// TIA Portal V18 export
DATA_BLOCK "WebDB"   // DB5
{ S7_Optimized_Access := 'FALSE' }
VERSION : 0.1
// stored: AutoNumber true, DBAccessibleFromOPCUA true, IsOnlyStoredInLoadMemory false, IsWriteProtectedInAS false
   VAR
      Enabled_Devices : Bool;   // Diagnostic value, necessary in step 3 (Check if system is ready); TRUE if OK;
      Ready_Devices : Bool;   // Diagnostic value, necessary in step 3 (Check if system is ready); TRUE if OK;
      Warning_Devices : Bool;   // Diagnostic value, necessary in step 3 (Check if system is ready); TRUE if OK;
      Fault_Devices : Bool;   // Diagnostic value, necessary in step 3 (Check if system is ready); TRUE if OK;
      diagMode { ExternalAccessible := 'False'; ExternalVisible := 'False'; ExternalWritable := 'False'} : UInt := 1;   // Diagnostic mode : 0
      myLADDR { ExternalAccessible := 'False'; ExternalVisible := 'False'; ExternalWritable := 'False'} : HW_ANY := 52;   // ID of CPUExecutUnit : 52 PLC ID: 64
      returnValue : Int;   // No error: 0
      CountDiagDetails : UInt;   // Should always be 0
      PLCDiag { S7_SetPoint := 'True'} : DIS;   // Read value of diagnostic
      Start_Machine : Bool;   // Button - Start Machine
      Stop_Machine : Bool;   // Button - Stop Machine
      Reset_error { ExternalAccessible := 'False'; ExternalVisible := 'False'; ExternalWritable := 'False'} : Bool;   // Button - Reset error after emergancy stop and other situation
      Stop_All_Axis : Bool;
      XInput : Struct
         EnableDrive : Bool;
         Stop : Bool;
         Halt : Bool;
         Brake : Bool;
         ResetFault : Bool;
         HMIAccessLocked : Bool;
         OPM : Int;   // Operating Mode ???
         StartTask : Bool;
         StartHoming : Bool;
         JogPos : Bool;
         JogNeg : Bool;
         TeachActValue : Bool;
         ClearRemPos : Bool;
         Relative : Bool;
         DeactivateStrokeLimit : Bool;
         ExecuteFunction : Bool;
         RecordNo : Int;
         SetFunctionNumber : Int;
         SetFunctionGroup : Int;
         SetValueVelocity : DInt := 20;
         SetValuePosition : DInt;
         SetValueForceRamp : DInt;
         SetValueForce : DInt;
         SetValueRotRamp : DInt;
         SetValueRotSpeed : DInt;
      END_STRUCT;
      XOutput : Struct
         DriveEnabled : Bool;
         Ready : Bool;
         Warning : Bool;
         Fault : Bool;
         SupplyVoltPresent : Bool;
         ControlFCT_HMI : Bool;
         StateOPM : Int;
         HaltNotActive : Bool;
         AckStart : Bool;
         MC : Bool;
         AckTeach : Bool;
         DriveMoving : Bool;
         DragError : Bool;
         StandStillControl : Bool;
         HomingValid : Bool;
         ActualRecordNo : Int;
         RC1 : Bool;
         RCC : Bool;
         VelocityLimitReached : Bool;
         StrokeLimitReached : Bool;
         FunctionIsActive : Bool;
         ActualFunctionNumber : Int;
         ActualFunctionGroup : Int;
         ActualPosition : DInt;
         ActualVelocity : DInt;
         ActualForce : DInt;
         ActualRotRamp : DInt;
         ActualRotSpeed : DInt;
      END_STRUCT;
      XAddOn1 : Struct
         XTargetRange : DInt := 1000;
         XTargetReached : Bool;
         XOverrange : Bool;
         Error_message_X : DInt;   // Number of error in DINT. Check error in CMMP documentation
         Restart_CMMO_X : Bool;   // Restart CMMP X controller
      END_STRUCT;
      YInput : Struct
         EnableDrive : Bool;
         Stop : Bool;
         Halt : Bool;
         Brake : Bool;
         ResetFault : Bool;
         HMIAccessLocked : Bool;
         OPM : Int;   // Operating Mode ???
         StartTask : Bool;
         StartHoming : Bool;
         JogPos : Bool;
         JogNeg : Bool;
         TeachActValue : Bool;
         ClearRemPos : Bool;
         Relative : Bool;
         DeactivateStrokeLimit : Bool;
         ExecuteFunction : Bool;
         RecordNo : Int;
         SetFunctionNumber : Int;
         SetFunctionGroup : Int;
         SetValueVelocity : DInt := 20;
         SetValuePosition : DInt;
         SetValueForceRamp : DInt;
         SetValueForce : DInt;
         SetValueRotRamp : DInt;
         SetValueRotSpeed : DInt;
      END_STRUCT;
      YOutput : Struct
         DriveEnabled : Bool;
         Ready : Bool;
         Warning : Bool;
         Fault : Bool;
         SupplyVoltPresent : Bool;
         ControlFCT_HMI : Bool;
         StateOPM : Int;
         HaltNotActive : Bool;
         AckStart : Bool;
         MC : Bool;
         AckTeach : Bool;
         DriveMoving : Bool;
         DragError : Bool;
         StandStillControl : Bool;
         HomingValid : Bool;
         ActualRecordNo : Int;
         RC1 : Bool;
         RCC : Bool;
         VelocityLimitReached : Bool;
         StrokeLimitReached : Bool;
         FunctionIsActive : Bool;
         ActualFunctionNumber : Int;
         ActualFunctionGroup : Int;
         ActualPosition : DInt;
         ActualVelocity : DInt;
         ActualForce : DInt;
         ActualRotRamp : DInt;
         ActualRotSpeed : DInt;
      END_STRUCT;
      YAddOn1 : Struct
         YTargetRange : DInt := 1000;
         YTargetReached : Bool;
         YOverrange : Bool;
         Error_message_Y : DInt;   // Number of error in DINT. Check error in CMMP documentation
         Restart_CMMO_Y : Bool;   // Restart CMMP Y controller
      END_STRUCT;
      Z1Input : Struct
         EnableDrive : Bool;
         Stop : Bool;
         Halt : Bool;
         Brake : Bool;
         ResetFault : Bool;
         HMIAccessLocked : Bool;
         OPM : Int;   // Operating Mode ???
         StartTask : Bool;
         StartHoming : Bool;
         JogPos : Bool;
         JogNeg : Bool;
         TeachActValue : Bool;
         ClearRemPos : Bool;
         Relative : Bool;
         DeactivateStrokeLimit : Bool;
         ExecuteFunction : Bool;
         RecordNo : Int;
         SetFunctionNumber : Int;
         SetFunctionGroup : Int;
         SetValueVelocity : DInt := 20;
         SetValuePosition : DInt;
         SetValueForceRamp : DInt;
         SetValueForce : DInt;
         SetValueRotRamp : DInt;
         SetValueRotSpeed : DInt;
      END_STRUCT;
      Z1Output : Struct
         DriveEnabled : Bool;
         Ready : Bool;
         Warning : Bool;
         Fault : Bool;
         SupplyVoltPresent : Bool;
         ControlFCT_HMI : Bool;
         StateOPM : Int;
         HaltNotActive : Bool;
         AckStart : Bool;
         MC : Bool;
         AckTeach : Bool;
         DriveMoving : Bool;
         DragError : Bool;
         StandStillControl : Bool;
         HomingValid : Bool;
         ActualRecordNo : Int;
         RC1 : Bool;
         RCC : Bool;
         VelocityLimitReached : Bool;
         StrokeLimitReached : Bool;
         FunctionIsActive : Bool;
         ActualFunctionNumber : Int;
         ActualFunctionGroup : Int;
         ActualPosition : DInt;
         ActualVelocity : DInt;
         ActualForce : DInt;
         ActualRotRamp : DInt;
         ActualRotSpeed : DInt;
      END_STRUCT;
      Z1AddOn1 : Struct
         Z1TargetRange : DInt := 1000;
         Z1TargetReached : Bool;
         Z1Overrange : Bool;
         Error_message_Z1 : DInt;   // Number of error in DINT. Check error in CMMO documentation
         Restart_CMMO_Z1 : Bool;   // Restart CMMO Z1 controller
      END_STRUCT;
      Z2Input : Struct
         EnableDrive : Bool;
         Stop : Bool;
         Halt : Bool;
         Brake : Bool;
         ResetFault : Bool;
         HMIAccessLocked : Bool;
         OPM : Int;   // Operating Mode ???
         StartTask : Bool;
         StartHoming : Bool;
         JogPos : Bool;
         JogNeg : Bool;
         TeachActValue : Bool;
         ClearRemPos : Bool;
         Relative : Bool;
         DeactivateStrokeLimit : Bool;
         ExecuteFunction : Bool;
         RecordNo : Int;
         SetFunctionNumber : Int;
         SetFunctionGroup : Int;
         SetValueVelocity : DInt := 20;
         SetValuePosition : DInt;
         SetValueForceRamp : DInt;
         SetValueForce : DInt;
         SetValueRotRamp : DInt;
         SetValueRotSpeed : DInt;
      END_STRUCT;
      Z2Output : Struct
         DriveEnabled : Bool;
         Ready : Bool;
         Warning : Bool;
         Fault : Bool;
         SupplyVoltPresent : Bool;
         ControlFCT_HMI : Bool;
         StateOPM : Int;
         HaltNotActive : Bool;
         AckStart : Bool;
         MC : Bool;
         AckTeach : Bool;
         DriveMoving : Bool;
         DragError : Bool;
         StandStillControl : Bool;
         HomingValid : Bool;
         ActualRecordNo : Int;
         RC1 : Bool;
         RCC : Bool;
         VelocityLimitReached : Bool;
         StrokeLimitReached : Bool;
         FunctionIsActive : Bool;
         ActualFunctionNumber : Int;
         ActualFunctionGroup : Int;
         ActualPosition : DInt;
         ActualVelocity : DInt;
         ActualForce : DInt;
         ActualRotRamp : DInt;
         ActualRotSpeed : DInt;
      END_STRUCT;
      Z2AddOn1 : Struct
         Z2TargetRange : DInt := 1000;
         Z2TargetReached : Bool;
         Z2Overrange : Bool;
         Error_message_Z2 : DInt;   // Number of error in DINT, Check error in CMMO documentation
         Restart_CMMO_Z2 : Bool;   // Restart CMMO Z2 controller
      END_STRUCT;
      Start_Roller : Bool;   // Set ON the rotations of the roller
      Stop_Roller : Bool;   // Reset OFF the rotations of the roller
      Output_Roller : Bool;
      SpreadParam : Struct
         spreadCycleYFirstPos : DInt;
         spreadCycleYSecondPos : DInt := 400000;
         spreadCycleYLastPos : DInt := 900000;
         Spread_BUSY : Bool;   // When spreading cycle is being executed - > TRUE
         Spread_DONE : Bool;   // Rising edge / When spreading cycle is done
         Spread_speed : DInt := 10;   // Value of speed (Y- axis) when the roller is above the printing bed
         Amount_of_layer : Int := 1;   // How many times do you want execute the spreading cycle ? How many powder layers do you want to spread ? Set value here.
         Spread_powder_stop : Bool;   // Spreading cycle - stop
         Spread_powder_execute : Bool;   // Spreading cycle - start / Don't forget set "Move_Feed" and "Move_Printing"
         Spread_Step_Z1 : DInt := 330;   // Relative movement / Set value / How much you want to up ?
         Spread_Step_Z2 : DInt := -300;   // Relative movement / How much you want to down ?
      END_STRUCT;
      Homing_all_axis : Bool;   // Press if you want execute homing for all axis
      SystemStatus : Struct   // System status: door sensor and emergency
         Emergency : Bool;   // Emergency button is active
         DoorSensor : Bool;
      END_STRUCT;
      Heater_ON : Bool;   // If you want to use the heater -> TRUE, if you don't want -> FALSE, Heater is activated during the spreading cycle
      PID_Heater_ON : Bool;   // If you want to use PID controller to control the temperature of powder - > TRUE , If the heater should be ON continuously -> FALSE, this option can be only activated when "Heater_ON" is TRUE
      WeightFluidTank : UInt;   // Weight in Kg
      WeightWastTank : UInt;   // Weight in Kg
      Heater_Setpoint : Real;   // Heating Setpoint [%] - future -> [Celsius]
      Heater_Sensor : Real;
      Heater_PDL : Real := 100.0;   // Pulse Duration Limit [%] - future -> [Celsius] set by technician or engineer in charge, don't change
      CappingStationInput : Struct
         CSMoveUP : Bool;   // Move capping station to the top position
         CSMoveDOWN : Bool;   // Move capping station to the bottom
      END_STRUCT;
      CappingStationOuput : Struct
         CSPositionUP : Bool;   // Confirmation of the top position reached
         CSPositionDOWN : Bool;   // Confirmation of the bottom position reached
         CSPosition : UInt;   // Actual position reading based on an estimation
         CSXYMotionLock : Bool;   // Motion lock to prevent destroying mechanism with the moving parts
      END_STRUCT;
      RollerAdjustableInput : Struct
         Mode : Int;   // 0; 1; 2; 3;
         SetSpeed : Real;   // %
         Direction : Bool;   // CW; CCW;
         OffsetSpeed : DInt;   // In mm/s
      END_STRUCT;
      RollerAdjustableOutput : Struct
         RollerDirection : Bool;
         RollerLinearVelocity : DInt;   // Relative speed of the roller surface in relation to the printbed surface
         setpointRPM : Real;
         RollerSpeedRPM : Real;   // Roller RPM - Measured
      END_STRUCT;
      UVLampInput : Struct   // Control of the UV lamp from NOAH
         UVLampEnable : Bool;   // Enable control block
         UVLampMode : Int;   // Choose lamp mode
         UVLampONOFF : Bool;   // Turn UV lamp ON and OFF
         UVLampSetpoint : Real;   // To enable the lamp, minimum 1V output
         UVLampMaintenance : Int;   // Maintenance mode to skip some of the safety rules
      END_STRUCT;
      UVLampOutput : Struct   // Status of the UV lamp in the PLC
         UVLampEnabled : Bool;
         UVLampWorking : Bool;   // 1 if lamp is ON; 0 if lamp is OFF
         UVLampError : Bool;   // 1 if OK; 0 if ERROR;
         UVLampIntensity : Real;   // Control Voltage 0-10V;
         UVLampStatus : Int;   // N/A
      END_STRUCT;
      StacklightInput : Struct   // Control of the Stacklight from NOAH
         StacklightEnable : Bool;   // 0 - working; 1 OFF;
         StacklightMode : Int;   // 0 - default mode;
         NOAHColor : Int;   // 0 red; 1 yellow; 2 green
         NOAHConnected : Bool;   // Checking if the connection is working
         NOAHPrinting : Bool;   // For the next version
         NOAHPaused : Bool;   // For the next version
         NOAHFluidError : Bool;
         StacklightMaintenance : Int;   // For special comands from NOAH
      END_STRUCT;
      StacklightOutput : Struct   // Status of the Stacklight in the PLC
         StacklightStatus : Int;   // N/A
         StaklightError : Bool;   // N/A
         StacklightColor : Int;   // 0 red; 1 yellow; 2 green
         StacklightCTRL01 : Bool;   // 0 Red; 1 Orange or Green;
         StacklightCTRL02 : Bool;   // 0 Orange; 1 Green;
      END_STRUCT;
      NoGoZone01AxisControl : Struct   // Control of the NoGoZone with restricted access
         NoGoMotionLockXmove : Bool;
         NoGoMotionLockXjog : Bool;
         NoGoMotionLockYmove : Bool;
         NoGoMotionLockYjog : Bool;
         NoGoMotionLockZ1move : Bool;
         NoGoMotionLockZ1jog : Bool;
         NoGoMotionLockZ2move : Bool;
         NoGoMotionLockZ2jog : Bool;
         HomingPermissionX : Bool;
         HomingPermissionY : Bool;
         HomingPermissionZ1 : Bool;
         HomingPermissionZ2 : Bool;
         NoGoAlwaysOn : Bool;
      END_STRUCT;
      NoGoZone01Status : Struct   // Status of the NoGoZone with restricted access
         NoGoZone01Active : Bool;
         YouAreInNoGoZone01 : Bool;
         CollisionErrorNoGoZone01 : Bool;
      END_STRUCT;
      PrintingStatus : Struct   // Printing Status Input from NOAH
         InPrintStarted : Bool;   // Input from Noah if the print was started
         InPrintPaused : Bool;   // Input from Noah if the print was paused
         InPrintEnded : Bool;   // Input from Noah if the print was ended
         OutMissingLayerDetected : Bool;   // Missing Layer Detection From The PLC
      END_STRUCT;
   END_VAR
BEGIN
END_DATA_BLOCK
